TYPE ST_EL3773_InputSamples_Scaled :
STRUCT
// Inputs from EL3773
	aUL1 : ARRAY[1..cOversamples] OF LREAL;
	aUL2 : ARRAY[1..cOversamples] OF LREAL;
	aUL3 : ARRAY[1..cOversamples] OF LREAL;
	aIL1 : ARRAY[1..cOversamples] OF LREAL;
	aIL2 : ARRAY[1..cOversamples] OF LREAL;
	aIL3 : ARRAY[1..cOversamples] OF LREAL;
END_STRUCT
END_TYPE

(* stored: Version 1.1.0.1, ProductVersion 3.1.4024.12
   DUT ST_EL3773_InputSamples_Scaled: Id {4c70ae45-8a2a-4da1-b1ba-ed18302a4175} *)
